{attribute 'qualified_only'}
VAR_GLOBAL CONSTANT
END_VAR

(* stored: Version 1.1.0.1, ProductVersion 3.1.4024.16
   GVL Param: Id {f89724df-0d6e-47a7-9e57-36c1a7871e93}, ParameterList True *)
